{attribute addProperty BoxType "EL3773-0000-0019"}
{attribute addProperty Id "I3_SamplesAT %I*ARRAY [0..9] OF INT16020"}
{attribute addProperty CRC "1727899378"}
{attribute addProperty SizeInBites "160"}
{attribute addProperty SizeInBytes "20"}
TYPE L3_Current_Samples_66FDA6F2 :
STRUCT
	{attribute addProperty Name "I3_Samples"}
	I3_Samples AT %I* : ARRAY [0..9] OF INT;
END_STRUCT
END_TYPE

(* stored: Version 1.2.0.0, ProductVersion 3.1.4024.9
   DUT L3_Current_Samples_66FDA6F2: Id {39a849e9-bbc2-4888-baaa-efdcc47c42c4} *)
